SUBAPPLICATION MERGE_SWITCH_1_QXA_OPC (* 1-Richtungs-Ausgang: bestehendes IO-Test-Kommando (Remote-Subscribe) wird mit dem echten Funktions-Kommando (Remote-Subscribe) per AX_OR_2 zusammengefuehrt - IO-Test bleibt nutzbar. Ausgang treibt den physischen logiBUS-Kanal UND meldet seinen Zustand sowohl an die bestehende IO-Test-Ueberwachung als auch an die echte Funktions-Rueckmeldung (z.B. GreenWhiteBackground am SoftKey) zurueck. Generisch fuer jeden einfachen (nicht doppelwirkenden) Ausgang mit Bedienung von einem Modul ohne eigenes VT - fuer doppelwirkende Aktoren (Links/Rechts, Auf/Ab) stattdessen ILOCK_SWITCH_2_QXA_OPC verwenden. *)
  (* Standard: 61499-2; Description: Copyright (c) 2026 Meisterschulen am Ostbahnhof This program and the accompanying materials are made available under the terms of the Eclipse Public License 2.0 which is available at https://www.eclipse.org/legal/epl-2.0/ SPDX-License-Identifier: EPL-2.0 *)
  (* Version 1.0, 2026-09-07, Franz Höpfinger, Meisterschulen am Ostbahnhof, initial API and implementation and/or initial documentation - 1-Richtungs-Analogon zu ILOCK_SWITCH_2_QXA_OPC (ohne Interlock/Schutzzeit, da keine Gegenrichtung zu schuetzen ist) *)
  PACKAGE MyLib::sys;
  IMPORT logiBUS::io::DQ::logiBUS_DO;
  IMPORT logiBUS::io::DQ::logiBUS_DO_S;
  (* Documentation:
  1-Richtungs-Ausgang: IO-Test ODER echtes Kommando (Pegel-ODER)
   1-Richtungs-Analogon zu ILOCK_SWITCH_2_QXA_OPC - fuer einfache Ausgaenge (z.B. Blitzlicht, Beleuchtung) ohne Gegenrichtung, die deshalb auch keinen Interlock/keine Schutzzeit brauchen. Bestehendes IO-Test-Kommando UND echtes Funktions-Kommando (SoftKey/AUX, per Softkey_Aux_IXA_TO_Remote_WRITE_BG_OPC auf dem Bedienmodul) werden per AX_OR_2 zusammengefuehrt und treiben gemeinsam den physischen Ausgang.
   Der resultierende Zustand wird auf ZWEI eigene, vom jeweiligen Kommando-Knoten getrennte Knoten zurueckgemeldet - ID_TEST_WRITE (fuer die bestehende IO-Diag-Anzeige) und ID_WRITE (fuer die echte Funktions-Rueckmeldung, z.B. Hintergrundfarbe am SoftKey). Kommando- und Status-Knoten duerfen sich NIE denselben OPC-UA-Knoten teilen, sonst liest die eigene Subscribe den eigenen Publish-Echo als neuen Befehl und der Ausgang haengt fest (siehe OPC_UA_VERNETZUNG.md Punkt 10+11).
  *)
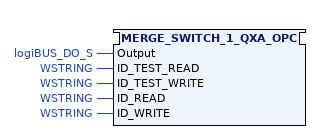
  VAR_INPUT
    Output : logiBUS::io::DQ::logiBUS_DO_S := logiBUS_DO::Invalid; (* Physischer Ausgang *)
    ID_TEST_READ : WSTRING; (* Bestehende IO-Test-Subscribe-Adresse (z.B. STG5_Q0x_READ) *)
    ID_TEST_WRITE : WSTRING; (* Bestehende IO-Test-Publish-Adresse (z.B. STG5_Q0x_WRITE) - EIGENER Knoten, NICHT ID_TEST_READs Knoten (sonst Selbstrueckkopplung/Latch, siehe OPC_UA_VERNETZUNG.md Punkt 10+11) *)
    ID_READ : WSTRING; (* Echtes Funktions-Kommando (Subscribe) *)
    ID_WRITE : WSTRING; (* Echte Funktions-Rueckmeldung (Publish) - EIGENER Knoten, NICHT ID_READs Knoten *)
  END_VAR
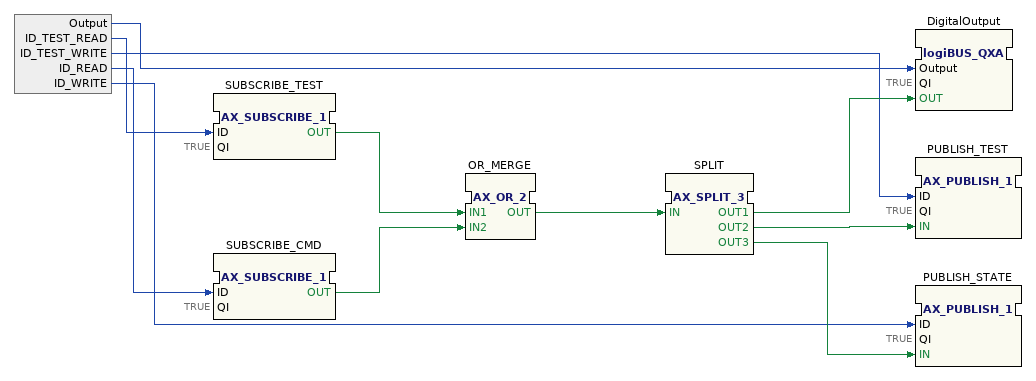
  FBS
    SUBSCRIBE_TEST : adapter::net::AX_SUBSCRIBE_1(QI := TRUE);
    SUBSCRIBE_CMD : adapter::net::AX_SUBSCRIBE_1(QI := TRUE);
    OR_MERGE : adapter::booleanOperators::AX_OR_2;
    DigitalOutput : logiBUS::io::DQ::logiBUS_QXA(QI := TRUE);
    SPLIT : adapter::events::unidirectional::AX_SPLIT_3;
    PUBLISH_TEST : adapter::net::AX_PUBLISH_1(QI := TRUE);
    PUBLISH_STATE : adapter::net::AX_PUBLISH_1(QI := TRUE);
  END_FBS
  DATA_CONNECTIONS
    ID_TEST_READ TO SUBSCRIBE_TEST.ID;
    ID_READ TO SUBSCRIBE_CMD.ID;
    Output TO DigitalOutput.Output;
    ID_TEST_WRITE TO PUBLISH_TEST.ID;
    ID_WRITE TO PUBLISH_STATE.ID;
  END_CONNECTIONS
  ADAPTER_CONNECTIONS
    SUBSCRIBE_TEST.OUT TO OR_MERGE.IN1;
    SUBSCRIBE_CMD.OUT TO OR_MERGE.IN2;
    OR_MERGE.OUT TO SPLIT.IN;
    SPLIT.OUT1 TO DigitalOutput.OUT;
    SPLIT.OUT2 TO PUBLISH_TEST.IN;
    SPLIT.OUT3 TO PUBLISH_STATE.IN;
  END_CONNECTIONS
END_SUBAPPLICATION
